// TIA Portal project "limit-switch" (V16)

(* hardware
DEVICE "S7-1200 station_1"  S7-1200 Station
   slot 0: "Rack_0"  S7-1200 Rack  Rack  V1.0
   slot 1: "PLC_1"  CPU 1212C AC/DC/Rly  6ES7 212-1BE40-0XB0  V4.4
*)

// ===== PLC "PLC_1"  CPU 1212C AC/DC/Rly =====

VAR_GLOBAL   // PLC tag table "Default tag table"
   "start" AT %I0.0 : Bool;
   "stop" AT %I0.1 : Bool;
   "LS1" AT %I0.2 : Bool;
   "LS2" AT %I0.3 : Bool;
   "LS3" AT %I0.4 : Bool;
   "km1" AT %Q0.0 : Bool;
   "km2" AT %Q0.1 : Bool;
   "Tag_1" AT %M0.0 : Bool;
END_VAR

ORGANIZATION_BLOCK "Main"   // OB1, LAD, ProgramCycle
TITLE = "Main Program Sweep (Cycle)"
{ S7_Optimized_Access := 'TRUE' }
VERSION : 0.1
   VAR_INPUT
      Initial_Call : Bool;   // Initial call of this OB
      Remanence : Bool;   // =True, if remanent data are available
   END_VAR
BEGIN

REGION Network 1
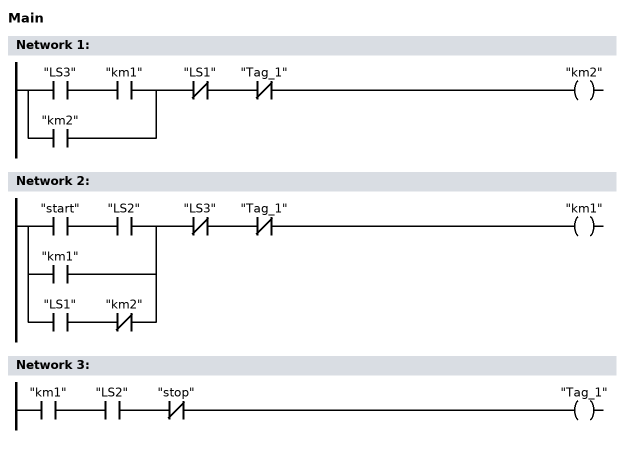
   RUNG wire#powerrail
      Contact( "LS3" )
      Contact( "km1" )
      wire#w1
      I_Contact( "LS1" )
      I_Contact( "Tag_1" )
      Coil( "km2" )
   END_RUNG
   RUNG wire#powerrail
      Contact( "km2" )
   END_RUNG wire#w1
   // the same network as SCL:
   "km2" := (("LS3" AND "km1") OR "km2") AND NOT "LS1" AND NOT "Tag_1";
END_REGION

REGION Network 2
   RUNG wire#powerrail
      Contact( "start" )
      Contact( "LS2" )
      wire#w1
      I_Contact( "LS3" )
      I_Contact( "Tag_1" )
      Coil( "km1" )
   END_RUNG
   RUNG wire#powerrail
      Contact( "km1" )
   END_RUNG wire#w1
   RUNG wire#powerrail
      Contact( "LS1" )
      I_Contact( "km2" )
   END_RUNG wire#w1
   // the same network as SCL:
   "km1" := (("start" AND "LS2") OR "km1" OR ("LS1" AND NOT "km2")) AND NOT "LS3" AND NOT "Tag_1";
END_REGION

REGION Network 3
   RUNG wire#powerrail
      Contact( "km1" )
      Contact( "LS2" )
      I_Contact( "stop" )
      Coil( "Tag_1" )
   END_RUNG
   // the same network as SCL:
   "Tag_1" := "km1" AND "LS2" AND NOT "stop";
END_REGION
END_ORGANIZATION_BLOCK